// TIA Portal V17 export
// export: Created 2022-04-06T07:28:41.2518447Z, ExportSetting WithDefaults, DisplayName Totally Integrated Automation Portal, DisplayVersion V17, DisplayName TIA Portal Openness, DisplayVersion V17, DisplayName TIA Portal Version Control Interface, DisplayVersion V17, DisplayName TIA Portal Test Suite Advanced, DisplayVersion V17, DisplayName SINAMICS Startdrive Advanced, DisplayVersion V17, DisplayName SINAMICS Startdrive G130, G150, S120, S150, SINAMICS MV, S210, DisplayVersion V17, DisplayName SINAMICS Startdrive G110M, G120, G120C, G120D, G120P, G115D, DisplayVersion V17, DisplayName STEP 7 Professional, DisplayVersion V17, DisplayName STEP 7 Safety, DisplayVersion V17, DisplayName WinCC Advanced / Unified PC, DisplayVersion V17
TYPE "LAxisCtrl_typeHoming"
TITLE = LAxisCtrl_typeHoming
// Support: tech.team.motioncontrol@siemens.com
// stored: IsFailsafeCompliant false
   STRUCT
      position : LReal := 0.0;   // The specified value is used according to the selected "Mode"
      mode : Int := 0;   // Operation mode; 0: Direct homing (absolute); 1: Direct homing (relative); 2: Passive homing (without reset); 3: Active homing; 5: Active homing (Position parameter has no effect); 6: Absolute encoder adjustment (relative); 7: Absolute encoder adjustment (absolute); 8:Passive homing ; 9: Abort passive homing; 10: Passive homing (Position parameter has no effect); 11: Set setpoint position (absolute); 12: Shift the setpoint position (relative)
      extendedMode : DInt := -1;   // -1: No extended homing mode (parameter "mode" is effective); 0: Homing on fixed stop; 1: Homing on fixed stop with moving out of clamping
      extendedModeTorqueLimit : LReal := 0.0;   // Value of the torque/force for extended homing mode
   END_STRUCT;
END_TYPE
